{attribute 'qualified_only'}
VAR_GLOBAL
	Status: BOOL;
	No: INT;
	Target_Pos_Moving: BOOL;
	Motion_Start: BOOL;
	Axis02_Work_Wait: BOOL;
	Press_Start: BOOL;
	Axis04_Torque_Controll: BOOL;
	Axis04_Wait_Pos_Moving: BOOL;
	All_Axis_Wait_Pos_Moving: BOOL;
	Work_Comp_Target_Pos_Moving: BOOL;
	All_Initial: BOOL;
	Axis02_Stop: BOOL;
	Z_Press_Start: BOOL;
	Force_Gear_Out: BOOL;   // 실패 abort 시 X축 gear-out 강제 (→ Axis02_Command MC_GearOut.Execute OR 입력)
END_VAR

(* stored: Version 1.1.0.1, ProductVersion 3.1.4024.15
   GVL GVL_Motion_Step: Id {0a3874d6-417c-4b69-a211-08b3ae03d94c} *)
